PROGRAM prgPersData
VAR
	fbPersData			: FB_WritePersistentData_CX51x0; 
END_VAR

fbPersData(
	eSaveModeData:= eUSVSaveMode.eSaveWhenPowerfail, 
	bLoadPersistentDataOk=> , 
	bPowerFailDetect=> , 
	bError=> , 
	bySaveProcess=> , 
	dwStorageLast24h=> , 
	udiErrorCode=> );

END_PROGRAM

(* stored: Version 1.1.0.1, ProductVersion 3.1.4024.9
   POU prgPersData: Id {f6f2047a-9d21-49b4-aeb3-b15e7685ac62}, SpecialFunc None *)
